// TIA Portal V18 export
DATA_BLOCK "PLC8_910A4_8DI_8DO_DI_Vars"   // DB11071
{ S7_Optimized_Access := 'FALSE' }
VERSION : 0.1
// stored: AutoNumber false, DBAccessibleFromOPCUA true, IsOnlyStoredInLoadMemory false, IsWriteProtectedInAS false
   VAR
      DI1 : "UDT_DIadv";   // AHU F Аварія ККБ
      DI2 : "UDT_DIadv";   // AHU F Ін. 1- ст. ККБ
      DI3 : "UDT_DIadv";   // AHU F Ін. 2- ст. ККБ
      DI4 : "UDT_DIadv";   // Резерв
      DI5 : "UDT_DIadv";   // Резерв
      DI6 : "UDT_DIadv";   // Резерв
      DI7 : "UDT_DIadv";   // Резерв
      DI8 : "UDT_DIadv";   // Резерв
   END_VAR
BEGIN
   DI4.cFuncSystemID := 100;
   DI4.cFuncVar := 7;
   DI5.cFuncSystemID := 1;
   DI5.cFuncVar := 17;
   DI6.cFuncSystemID := 1;
   DI6.cFuncVar := 18;
   DI7.cFuncSystemID := 1;
   DI7.cFuncVar := 16;
END_DATA_BLOCK
